RoomTemp_205();
TempAdjust_205();
FilterSign_205();
FilterSignReset_205();
RemoteControlStart_205();

RemoteControlTempAdjust_205();












StartStopCommand_206();
StartStopStatus_206();
Alarm_206();
MalfunctionCode_206();




RoomTemp_206();
TempAdjust_206();
FilterSign_206();
FilterSignReset_206();
RemoteControlStart_206();

RemoteControlTempAdjust_206();












StartStopCommand_207();
StartStopStatus_207();
Alarm_207();
MalfunctionCode_207();




RoomTemp_207();
TempAdjust_207();
FilterSign_207();
FilterSignReset_207();
RemoteControlStart_207();

RemoteControlTempAdjust_207();












StartStopCommand_208();
StartStopStatus_208();
Alarm_208();
MalfunctionCode_208();




RoomTemp_208();
TempAdjust_208();
FilterSign_208();
FilterSignReset_208();
RemoteControlStart_208();

RemoteControlTempAdjust_208();












StartStopCommand_209();
StartStopStatus_209();
Alarm_209();
MalfunctionCode_209();




RoomTemp_209();
TempAdjust_209();
FilterSign_209();
FilterSignReset_209();
RemoteControlStart_209();

RemoteControlTempAdjust_209();












StartStopCommand_210();
StartStopStatus_210();
Alarm_210();
MalfunctionCode_210();




RoomTemp_210();
TempAdjust_210();
FilterSign_210();
FilterSignReset_210();
RemoteControlStart_210();

RemoteControlTempAdjust_210();












StartStopCommand_211();
StartStopStatus_211();
Alarm_211();
MalfunctionCode_211();




RoomTemp_211();
TempAdjust_211();
FilterSign_211();
FilterSignReset_211();
RemoteControlStart_211();

RemoteControlTempAdjust_211();












StartStopCommand_214();
StartStopStatus_214();
Alarm_214();
MalfunctionCode_214();




RoomTemp_214();
TempAdjust_214();
FilterSign_214();
FilterSignReset_214();
RemoteControlStart_214();

RemoteControlTempAdjust_214();












StartStopCommand_215();
StartStopStatus_215();
Alarm_215();
MalfunctionCode_215();




RoomTemp_215();
TempAdjust_215();
FilterSign_215();
FilterSignReset_215();
RemoteControlStart_215();

RemoteControlTempAdjust_215();












StartStopCommand_216();
StartStopStatus_216();
Alarm_216();
MalfunctionCode_216();




RoomTemp_216();
TempAdjust_216();
FilterSign_216();
FilterSignReset_216();
RemoteControlStart_216();

RemoteControlTempAdjust_216();












StartStopCommand_224();
StartStopStatus_224();
Alarm_224();
MalfunctionCode_224();




RoomTemp_224();
TempAdjust_224();
FilterSign_224();
FilterSignReset_224();
RemoteControlStart_224();

RemoteControlTempAdjust_224();












StartStopCommand_225();
StartStopStatus_225();
Alarm_225();
MalfunctionCode_225();




RoomTemp_225();
TempAdjust_225();
FilterSign_225();
FilterSignReset_225();
RemoteControlStart_225();

RemoteControlTempAdjust_225();












StartStopCommand_226();
StartStopStatus_226();
Alarm_226();
MalfunctionCode_226();




RoomTemp_226();
TempAdjust_226();
FilterSign_226();
FilterSignReset_226();
RemoteControlStart_226();

RemoteControlTempAdjust_226();












StartStopCommand_228();
StartStopStatus_228();
Alarm_228();
MalfunctionCode_228();




RoomTemp_228();
TempAdjust_228();
FilterSign_228();
FilterSignReset_228();
RemoteControlStart_228();

RemoteControlTempAdjust_228();












StartStopCommand_229();
StartStopStatus_229();
Alarm_229();
MalfunctionCode_229();




RoomTemp_229();
TempAdjust_229();
FilterSign_229();
FilterSignReset_229();
RemoteControlStart_229();

RemoteControlTempAdjust_229();












StartStopCommand_230();
StartStopStatus_230();
Alarm_230();
MalfunctionCode_230();




RoomTemp_230();
TempAdjust_230();
FilterSign_230();
FilterSignReset_230();
RemoteControlStart_230();

RemoteControlTempAdjust_230();












StartStopCommand_231();
StartStopStatus_231();
Alarm_231();
MalfunctionCode_231();




RoomTemp_231();
TempAdjust_231();
FilterSign_231();
FilterSignReset_231();
RemoteControlStart_231();

RemoteControlTempAdjust_231();












StartStopCommand_232();
StartStopStatus_232();
Alarm_232();
MalfunctionCode_232();




RoomTemp_232();
TempAdjust_232();
FilterSign_232();
FilterSignReset_232();
RemoteControlStart_232();

RemoteControlTempAdjust_232();












StartStopCommand_233();
StartStopStatus_233();
Alarm_233();
MalfunctionCode_233();




RoomTemp_233();
TempAdjust_233();
FilterSign_233();
FilterSignReset_233();
RemoteControlStart_233();

RemoteControlTempAdjust_233();












StartStopCommand_234();
StartStopStatus_234();
Alarm_234();
MalfunctionCode_234();




RoomTemp_234();
TempAdjust_234();
FilterSign_234();
FilterSignReset_234();
RemoteControlStart_234();

RemoteControlTempAdjust_234();












StartStopCommand_241();
StartStopStatus_241();
Alarm_241();
MalfunctionCode_241();




RoomTemp_241();
TempAdjust_241();
FilterSign_241();
FilterSignReset_241();
RemoteControlStart_241();

RemoteControlTempAdjust_241();












CL_Rejection_000();
SystemForcedOff_000();
CL_Rejection_064();
SystemForcedOff_064();
CL_Rejection_128();
SystemForcedOff_128();
CL_Rejection_192();
SystemForcedOff_192();

END_FUNCTION_BLOCK

(* stored: Version 1.1.0.1, ProductVersion 3.1.4024.14
   POU FB_BACnet_DAIKIN_MasterStation_III_No_6: Id {4c7e3e93-0451-409a-8978-4502b3736a48}, SpecialFunc None *)
